FUNCTION_BLOCK FlushingManager (* CAT Function Block Type *)
  (* Standard: 61499-2 *)
  (* Version 0.0, 6/21/2026, Schneider Electric, template *)
  PACKAGE SE.Nereda;
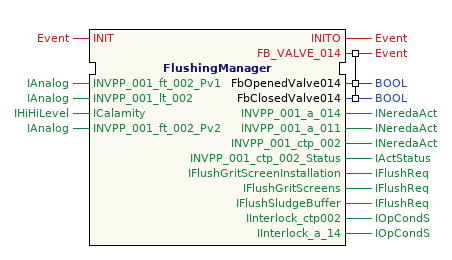
  EVENT_INPUT
    INIT;
  END_EVENT
  EVENT_OUTPUT
    INITO;
    FB_VALVE_014 WITH FbOpenedValve014, FbClosedValve014;
  END_EVENT
  VAR_OUTPUT
    FbOpenedValve014 : BOOL;
    FbClosedValve014 : BOOL;
  END_VAR
  SOCKETS
    INVPP_001_ft_002_Pv1 : IAnalog;
    INVPP_001_lt_002 : IAnalog;
    ICalamity : IHiHiLevel;
  END_SOCKETS
  SOCKETS
    INVPP_001_ft_002_Pv2 : IAnalog; (* Process value (range considered) interface adapter *)
  END_SOCKETS
  PLUGS
    INVPP_001_a_014 : INeredaAct;
    INVPP_001_a_011 : INeredaAct;
    INVPP_001_ctp_002 : INeredaAct;
    INVPP_001_ctp_002_Status : IActStatus;
  END_PLUGS
  PLUGS
    IFlushGritScreenInstallation : IFlushReq;
    IFlushGritScreens : IFlushReq;
    IFlushSludgeBuffer : IFlushReq;
    IInterlock_ctp002 : IOpCondS; (* Condition summary chain output to downstream block *)
    IInterlock_a_14 : IOpCondS; (* Condition summary chain output to downstream block *)
  END_PLUGS
  (* 01 - FUNCTIONNAL INPUT INTERFACE *)
  (* 00 - INITIALIZATION *)
  (* 05 - LOGIC *)
  (* 06 - HMI INTERFACE *)
  (* 03 - FIELD INTERFACE *)
  (* Eflluent Pump & Valves Conditions *)
  (* 02 - FUNCTIONNAL OUTPUT INTERFACE *)
  (* Eflluent Pump & Valves Control *)
  (* Flushing Control & Selector *)
  (* Interlock *)
  FBS
    IThis : FlushingManager_HMI(QI := TRUE);
    NVPP_001_lt_002_Status : decodeStatus; {SET_ATTRIBUTE(Configuration.Component.HideUnusedPorts, )}
    NVPP_001_ft_002_Status : decodeStatus; {SET_ATTRIBUTE(Configuration.Component.HideUnusedPorts, )}
    EffluentPumpCdts : EffluentCdt(pin_D80C7C0ABBECCDAB := 'Effluent Start Conditions', pin_386488C1B3EEC32A := 'Effluent Stop Conditions', pin_AD4F1D04748929A2 := 'Start Pump - Effluent', pin_E55C299A5BCFE2A5 := 'NVPP 001 a-- 011 is Available', pin_4F5AA965534A9167 := 'NVPP 001 a-- 014 is Available', pin_D8438E8592CCBB68 := 'Effluent Pump is Ready', pin_F9CA602A9987631B := 'Stop Pump - Effluent', pin_D946781DFBE190E0 := 'Hight Hight Level - Calamity', pin_EDFD852BF7F500FC := '', pin_2D24E9AB41BE5BDB := FALSE, pin_2F47EB70426E0A5E := 'Low Level - Effluent');
    EffluentControl : FlushingManagerEffluent;
    PumpCmd : boolValueChanged;
    Valve11Cmd : boolValueChanged;
    Valve14Cmd : boolValueChanged;
    FlushControlSelector : FlushSelector;
    PID_CTP_002 : PID; {SET_ATTRIBUTE(Configuration.Component.HideUnusedPorts, )}
    SpeedSp : SELECT_1513674226BA3DDCB(IN1 := 0.0); {SET_ATTRIBUTE(Configuration.GenericFBType.InterfaceParams, Runtime.Standard#CNT:=3;SELECT:INT;IN${CNT$}:REAL)}
    SpeedSpSmooth : RealValueChanged;
    DelayFlowAlarm : DelayedActive(pin_4E076A4928A0DFEF := TRUE, pin_1CE054BDD0AD4DEB := T#1m);
    LowLowFlow : AND_88A3DD8EC65DD11C; {SET_ATTRIBUTE(Configuration.GenericFBType.InterfaceParams, Runtime.Standard#CNT:=2;OUT:BOOL)}
    ResetBtns : RESET_BTNs;
    LowLowFlow_ctp002 : ilckCondItem(CondCause := Active1);
    HighHighLevel_Calamity : ilckCondItem(CondCause := Active1);
    HighHighCalamity : OR_88A3DD8EC65DD11C; {SET_ATTRIBUTE(Configuration.GenericFBType.InterfaceParams, Runtime.Standard#CNT:=2;OUT:BOOL)}
    HighHighLevel_Calamity1 : ilckCondItem(CondCause := Active1);
    HiHiCalamityAndPumpStopped : AND_88A3DD8EC65DD11C; {SET_ATTRIBUTE(Configuration.GenericFBType.InterfaceParams, Runtime.Standard#CNT:=2;OUT:BOOL)}
    PIDISc : PID_Manager;
    PumpCtp002 : BOOL2INT;
    Valve11 : BOOL2INT;
    Valve14 : BOOL2INT;
    FlushFlowSp_Select : FlushFlowSpManager;
    SpeedSp1 : SpeedSpFlowSensorFail;
    StartStopCdts : StartStopSpPv;
    LowLevel_Effluent : ilckCondItem(CondCause := Active1);
    Eff : RetriggerEvent(pin_FDD5DC24A8674AF6 := T#1s, pin_CFF51EFF0A91DC53 := 3);
  END_FBS
  EVENT_CONNECTIONS
    INVPP_001_lt_002.REQ_STATUS TO NVPP_001_lt_002_Status.REQ;
    INVPP_001_ft_002_Pv1.REQ_STATUS TO NVPP_001_ft_002_Status.REQ;
    Valve11Cmd.CNF TO Valve14Cmd.REQ;
    PID_CTP_002.CNF TO SpeedSp1.B5D6B08FA2666F02;
    NVPP_001_ft_002_Status.CNF TO LowLowFlow.REQ;
    LowLowFlow.CNF TO LowLowFlow_ctp002.REQ;
    HighHighCalamity.CNF TO HighHighLevel_Calamity.REQ;
    HighHighCalamity.CNF TO HiHiCalamityAndPumpStopped.REQ;
    HiHiCalamityAndPumpStopped.CNF TO HighHighLevel_Calamity1.REQ;
    NVPP_001_lt_002_Status.CNF TO StartStopCdts.19B0F962D4DCEDE2;
    PIDISc.CE80458C9D5EF15A TO INITO;
    ICalamity.15126F43E529BB4F TO StartStopCdts.19B0F962D4DCEDE2;
    ICalamity.15126F43E529BB4F TO HighHighCalamity.REQ;
    INVPP_001_a_011.CC753684FA882790 TO StartStopCdts.19B0F962D4DCEDE2;
    INVPP_001_a_014.CC753684FA882790 TO StartStopCdts.19B0F962D4DCEDE2;
    INVPP_001_ctp_002.CC753684FA882790 TO StartStopCdts.19B0F962D4DCEDE2;
    LowLowFlow.CNF TO StartStopCdts.19B0F962D4DCEDE2;
    EffluentPumpCdts.144BD964598CDC30 TO FlushControlSelector.6017B517BF713340;
    EffluentPumpCdts.E74FDFC5C9E17061 TO FlushControlSelector.9AFE71761EEDAA8D;
    EffluentControl.9CA068A916565A8E TO FlushControlSelector.734658F2C0A63384;
    INVPP_001_a_014.9CD053F8408797ED TO FlushControlSelector.8B5DB71997573DCB;
    INVPP_001_ctp_002.9CD053F8408797ED TO FlushControlSelector.C5600474CE829544;
    FlushControlSelector.F39EC8FC8C54BE8A TO PIDISc.INIT;
    FlushControlSelector.542E28C8E8F931AD TO EffluentControl.D2EC16313245450D;
    EffluentPumpCdts.144BD964598CDC30 TO Eff.2BC1963D96179493;
    INVPP_001_ctp_002.9CD053F8408797ED TO EffluentControl.4EF158ED5622E267;
    SpeedSpSmooth.93AE3729A9342678 TO EffluentControl.5683EF263AD86A9D;
    INVPP_001_ctp_002.F846995A4121D865 TO EffluentControl.676E3CF38C403777;
    INVPP_001_ctp_002.CC753684FA882790 TO EffluentControl.23B08E337BF80FCD;
    INVPP_001_a_011.9CD053F8408797ED TO EffluentControl.17EF565317C21577;
    INVPP_001_a_014.9CD053F8408797ED TO EffluentControl.17EF565317C21577;
    INVPP_001_a_011.CC753684FA882790 TO EffluentControl.968F0D58B28B83A2;
    INVPP_001_a_014.CC753684FA882790 TO EffluentControl.968F0D58B28B83A2;
    EffluentControl.C3A69DB7F9EE9593 TO PumpCmd.REQ;
    EffluentControl.91BAE91D4E0C293C TO SpeedSp.REQ;
    EffluentControl.7C8478AB3E0AC40C TO Valve11Cmd.REQ;
    PumpCmd.CHD TO PumpCtp002.DD5870AA881150BB;
    Valve11Cmd.CHD TO Valve11.DD5870AA881150BB;
    PumpCtp002.6FC99A5BD1C38561 TO INVPP_001_ctp_002.0F1CDF9A9B4A227A;
    Valve11.6FC99A5BD1C38561 TO INVPP_001_a_011.0F1CDF9A9B4A227A;
    Valve14Cmd.CHD TO Valve14.DD5870AA881150BB;
    Valve14.6FC99A5BD1C38561 TO INVPP_001_a_014.0F1CDF9A9B4A227A;
    SpeedSp.CNF TO SpeedSpSmooth.77F8F9CFF707DAFF;
    SpeedSpSmooth.350834820611931F TO INVPP_001_ctp_002.1E00729184986247;
    INVPP_001_ctp_002.9CD053F8408797ED TO DelayFlowAlarm.C451626F7187F42D;
    DelayFlowAlarm.DDA64CDC00519DA4 TO LowLowFlow.REQ;
    INVPP_001_ctp_002.9CD053F8408797ED TO HiHiCalamityAndPumpStopped.REQ;
    INVPP_001_a_014.9CD053F8408797ED TO FB_VALVE_014;
    PumpCtp002.6FC99A5BD1C38561 TO FlushFlowSp_Select.11EFC538173604A5;
    FlushFlowSp_Select.8933B5415DF4ADE7 TO PIDISc.REQ;
    FlushControlSelector.D8AC545B32F4E4B1 TO FlushFlowSp_Select.11EFC538173604A5;
    FlushControlSelector.D6D518D93DB5C2EF TO FlushFlowSp_Select.11EFC538173604A5;
    INIT TO IThis.AABF4BC3AB55D4F4;
    EffluentControl.GRAPH TO IThis.19BBDF43E4547D8F;
    INVPP_001_lt_002.REQ TO IThis.19941705FB9296A7;
    ResetBtns.920962203CA54948 TO IThis.D3057844E55CD2A1;
    FlushFlowSp_Select.8933B5415DF4ADE7 TO IThis.8FC64887EAD50F1F;
    FlushControlSelector.F39EC8FC8C54BE8A TO IThis.8E2191486483827C;
    IThis.67A10949F5B1AAAB TO EffluentPumpCdts.7689825C23C7E3C1;
    IThis.6F082D2834F78A1D TO SpeedSp.REQ;
    IThis.6F082D2834F78A1D TO EffluentControl.5683EF263AD86A9D;
    IThis.6F082D2834F78A1D TO FlushFlowSp_Select.11EFC538173604A5;
    IThis.B91C4BB13E300945 TO DelayFlowAlarm.C451626F7187F42D;
    IThis.B91C4BB13E300945 TO ResetBtns.AB695E9A35A20E19;
    INVPP_001_ctp_002.9CD053F8408797ED TO INVPP_001_ctp_002_Status.14377629A1F197A9;
    INVPP_001_ctp_002.F846995A4121D865 TO INVPP_001_ctp_002_Status.03F1F1C982EE8DD5;
    SpeedSp1.1FEAADE7145F64BE TO SpeedSp.REQ;
    FlushFlowSp_Select.8933B5415DF4ADE7 TO SpeedSp1.B5D6B08FA2666F02;
    NVPP_001_ft_002_Status.CNF TO SpeedSp1.B5D6B08FA2666F02;
    INVPP_001_ft_002_Pv1.REQ TO SpeedSp1.B5D6B08FA2666F02;
    StartStopCdts.ED0F74C511AB6DA4 TO EffluentPumpCdts.C4A26A2931936C6C;
    INVPP_001_lt_002.REQ TO StartStopCdts.19B0F962D4DCEDE2;
    IThis.04EFE92AD3E2EC6F TO StartStopCdts.19B0F962D4DCEDE2;
    NVPP_001_lt_002_Status.CNF TO LowLevel_Effluent.REQ;
    StartStopCdts.ED0F74C511AB6DA4 TO EffluentControl.A6AE1F3C3DDAB3ED;
    EffluentControl.6EFEB49A6788B5F1 TO FlushControlSelector.8D39C417490F8630;
    Eff.4002AEF0814D09CF TO EffluentControl.D2EC16313245450D;
  END_CONNECTIONS
  DATA_CONNECTIONS
    INVPP_001_lt_002.Status TO NVPP_001_lt_002_Status.Status;
    INVPP_001_ft_002_Pv1.Status TO NVPP_001_ft_002_Status.Status;
    PID_CTP_002.Out TO SpeedSp1.4727B0C2E5DD09FB;
    NVPP_001_ft_002_Status.LoLoAlarm TO LowLowFlow.IN2;
    LowLowFlow.OUT TO LowLowFlow_ctp002.CondSignal;
    HighHighCalamity.OUT TO HighHighLevel_Calamity.CondSignal;
    HighHighCalamity.OUT TO HiHiCalamityAndPumpStopped.IN1;
    HiHiCalamityAndPumpStopped.OUT TO HighHighLevel_Calamity1.CondSignal;
    ICalamity.C818324478A2F205 TO EffluentPumpCdts.4E3CFAB7818DC81F;
    ICalamity.C818324478A2F205 TO HighHighCalamity.IN1;
    ICalamity.96B50ADF37756FFC TO HighHighCalamity.IN2;
    INVPP_001_a_011.8A8A07EFCDA1443C TO EffluentPumpCdts.4ED40FD24D2392DA;
    INVPP_001_a_014.8A8A07EFCDA1443C TO EffluentPumpCdts.504E64E2CDCF5D86;
    INVPP_001_ctp_002.8A8A07EFCDA1443C TO EffluentPumpCdts.9BB2492C130556E4;
    EffluentPumpCdts.5C1922DA22925005 TO EffluentControl.AA1E4914E0281BF0;
    EffluentPumpCdts.F6D4C156FD41491A TO FlushControlSelector.78178F9D457C2392;
    EffluentPumpCdts.D0AD8FB829A4C538 TO EffluentControl.A9552914234A38C8;
    EffluentControl.B2669975DEFA0F4B TO FlushControlSelector.09149020AC3B86F2;
    INVPP_001_a_014.7F6CC7FEB9223DF3 TO FlushControlSelector.7BBAF2BC16CFB2C2;
    INVPP_001_a_014.A8D6C4A1FDCCA991 TO FlushControlSelector.ECC93065B5CD842A;
    INVPP_001_ctp_002.B762734C094A7162 TO FlushControlSelector.826F35173E83E980;
    INVPP_001_ctp_002.D83B5BDEFA4D797C TO FlushControlSelector.1576446F424BF684;
    FlushControlSelector.ADCCD13610E10A0A TO EffluentControl.14C00E94AA0EC676;
    FlushControlSelector.B35E76E6FAFFAA0F TO EffluentControl.93BA244FC15A95D2;
    FlushControlSelector.62ABA25AB0F002B3 TO EffluentControl.CEB88DEF7656C277;
    EffluentControl.F43CD565BDEA3238 TO PumpCmd.Input;
    EffluentControl.9D2A006C760775DE TO SpeedSp.SELECT;
    EffluentControl.6EFD4A5711C4475D TO Valve11Cmd.Input;
    EffluentControl.CB32327038C02D58 TO Valve14Cmd.Input;
    PumpCmd.Output TO PumpCtp002.4573FC8F228EB71D;
    Valve11Cmd.Output TO Valve11.4573FC8F228EB71D;
    PumpCmd.Output TO PIDISc.RunPID;
    PumpCtp002.A6DEF5F9C27C1848 TO INVPP_001_ctp_002.710D7FC54EE3F35A;
    Valve11.A6DEF5F9C27C1848 TO INVPP_001_a_011.710D7FC54EE3F35A;
    Valve14Cmd.Output TO Valve14.4573FC8F228EB71D;
    Valve14.A6DEF5F9C27C1848 TO INVPP_001_a_014.710D7FC54EE3F35A;
    SpeedSp.OUT TO SpeedSpSmooth.25B5287A5784F3EC;
    SpeedSpSmooth.AA81B8787A42C5C8 TO INVPP_001_ctp_002.1BC103921BBFDA0B;
    SpeedSpSmooth.AA81B8787A42C5C8 TO EffluentControl.3FA96986981E6302;
    DelayFlowAlarm.614F3125208254F6 TO LowLowFlow.IN1;
    INVPP_001_ctp_002.B762734C094A7162 TO DelayFlowAlarm.19546B227DE05AED;
    INVPP_001_ctp_002.D83B5BDEFA4D797C TO HiHiCalamityAndPumpStopped.IN2;
    INVPP_001_ctp_002.D83B5BDEFA4D797C TO EffluentControl.EBEF47FDF1899A9D;
    INVPP_001_ctp_002.B762734C094A7162 TO EffluentControl.9A4D3046FA82643D;
    INVPP_001_ctp_002.790C5C3BA88E0AF5 TO EffluentControl.139BE6F177247521;
    INVPP_001_ctp_002.8A8A07EFCDA1443C TO EffluentControl.FA41194B6CC39C55;
    INVPP_001_a_011.7F6CC7FEB9223DF3 TO EffluentControl.FB13F72D51F6D51B;
    INVPP_001_a_011.A8D6C4A1FDCCA991 TO EffluentControl.C38A322B1C43C4CB;
    INVPP_001_a_011.8A8A07EFCDA1443C TO EffluentControl.1E5D925B1F83133E;
    INVPP_001_a_014.7F6CC7FEB9223DF3 TO EffluentControl.20DA1363D32524AA;
    INVPP_001_a_014.A8D6C4A1FDCCA991 TO EffluentControl.3F622CAF90E39F0D;
    INVPP_001_a_014.8A8A07EFCDA1443C TO EffluentControl.9F8A5F98C564BB8A;
    INVPP_001_a_014.7F6CC7FEB9223DF3 TO FbOpenedValve014;
    INVPP_001_a_014.A8D6C4A1FDCCA991 TO FbClosedValve014;
    FlushFlowSp_Select.971EA695F43B2153 TO PIDISc.Setpoint;
    FlushControlSelector.747E185B5CA3297F TO FlushFlowSp_Select.D809E32A9AAF4DB7;
    FlushControlSelector.EDD14476E52E5293 TO FlushFlowSp_Select.1897BC4B6F9EA603;
    FlushControlSelector.CD6EADF9443800B0 TO FlushFlowSp_Select.2AB2CCE4EBBC9F51;
    FlushControlSelector.6044BC15C4CDD531 TO FlushFlowSp_Select.C3A04AF8A83D4A53;
    EffluentControl.Grafcet TO IThis.E29FE2D1F8D2DF4E;
    INVPP_001_lt_002.Value TO IThis.BCC4B883F9323D16;
    INVPP_001_lt_002.ValueMax TO IThis.58584200CBBD6E38;
    INVPP_001_lt_002.ValueMin TO IThis.798C728313EBA85C;
    IThis.12A65F1451D1D9B3 TO FlushFlowSp_Select.7BDB52087F72217A;
    IThis.D8F7ACDB7A0724E5 TO SpeedSp.IN2;
    IThis.D8F7ACDB7A0724E5 TO EffluentControl.E8C11D2A68704996;
    IThis.DC82B89A4AA2A4B1 TO DelayFlowAlarm.45767490F5BA3A44;
    IThis.DC82B89A4AA2A4B1 TO ResetBtns.479D4538AEFD6EE1;
    FlushFlowSp_Select.971EA695F43B2153 TO IThis.0B7AEE3E216B973E;
    INVPP_001_ctp_002.D83B5BDEFA4D797C TO INVPP_001_ctp_002_Status.227987A2F0C6A825;
    INVPP_001_ctp_002.B762734C094A7162 TO INVPP_001_ctp_002_Status.D41A46B14EF7208D;
    INVPP_001_ctp_002.790C5C3BA88E0AF5 TO INVPP_001_ctp_002_Status.B9E42D72CEF16844;
    INVPP_001_ctp_002.7F6CC7FEB9223DF3 TO INVPP_001_ctp_002_Status.72E790857420193D;
    INVPP_001_ctp_002.A8D6C4A1FDCCA991 TO INVPP_001_ctp_002_Status.3A653A8838D163CA;
    INVPP_001_ctp_002.8A8A07EFCDA1443C TO INVPP_001_ctp_002_Status.9E0B44559326BEAF;
    SpeedSp1.87931CA83794BFFD TO SpeedSp.IN3;
    FlushFlowSp_Select.971EA695F43B2153 TO SpeedSp1.3BE251DFC2E7905D;
    NVPP_001_ft_002_Status.FailAlarm TO SpeedSp1.1C28FEF37A13F67F;
    INVPP_001_ft_002_Pv1.ValueMax TO SpeedSp1.75C86D8B7647050C;
    INVPP_001_ft_002_Pv1.ValueMin TO SpeedSp1.B08827D02DBBFA97;
    StartStopCdts.91B941F57B403772 TO EffluentPumpCdts.22A84A30EE8DD605;
    StartStopCdts.79A07DF8BE81D140 TO EffluentPumpCdts.9D55FD7AD1246DA2;
    INVPP_001_lt_002.Value TO StartStopCdts.DD34EA40290B8853;
    IThis.64BC44F5776D6899 TO StartStopCdts.DA9D6C0B442BDE8A;
    IThis.4B2868EB90D190BF TO StartStopCdts.1127B3C1A86C2C47;
    NVPP_001_lt_002_Status.LoAlarm TO LowLevel_Effluent.CondSignal;
    NVPP_001_lt_002_Status.LoAlarm TO EffluentPumpCdts.47969CBC2D520AAD;
    StartStopCdts.91B941F57B403772 TO EffluentControl.3D8856C8DB36F2F8;
    StartStopCdts.79A07DF8BE81D140 TO EffluentControl.78CF96B4B163341F;
    EffluentControl.E4F48AF8C7D3F120 TO FlushControlSelector.24006E258DC9A0B4;
    EffluentControl.FEB150FEE0F179E0 TO FlushControlSelector.66D1CC7B71A96F98;
  END_CONNECTIONS
  ADAPTER_CONNECTIONS
    INVPP_001_ft_002_Pv2 TO PID_CTP_002.IPv;
    HighHighLevel_Calamity.ICondChainOut TO IInterlock_ctp002;
    LowLevel_Effluent.ICondChainOut TO HighHighLevel_Calamity.ICondChainIn;
    HighHighLevel_Calamity1.ICondChainOut TO IInterlock_a_14;
    FlushControlSelector.A0C84BB872573E34 TO IFlushGritScreenInstallation;
    FlushControlSelector.FD4617D32B0C81DC TO IFlushGritScreens;
    FlushControlSelector.CF996F44144FB07A TO IFlushSludgeBuffer;
    PIDISc.FACD1DD4E791A86A TO PID_CTP_002.ISc;
    LowLowFlow_ctp002.ICondChainOut TO LowLevel_Effluent.ICondChainIn;
  END_CONNECTIONS
END_FUNCTION_BLOCK
